FUNCTION_BLOCK SENSOR_SIMULATOR_V2
  {SET_ATTRIBUTE(OpcUa, DEVICE.SENSOR)}
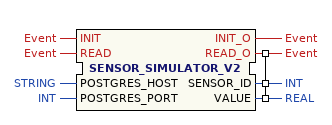
  EVENT_INPUT
    INIT;
    READ;
  END_EVENT
  EVENT_OUTPUT
    INIT_O;
    READ_O WITH VALUE, SENSOR_ID;
  END_EVENT
  VAR_INPUT
    POSTGRES_HOST : STRING; {SET_ATTRIBUTE(OpcUa, Constant)}
    POSTGRES_PORT : INT; {SET_ATTRIBUTE(OpcUa, Constant)}
  END_VAR
  VAR_OUTPUT
    SENSOR_ID : INT; {SET_ATTRIBUTE(OpcUa, Variable)}
    VALUE : REAL; {SET_ATTRIBUTE(OpcUa, Variable)}
  END_VAR
END_FUNCTION_BLOCK
